FUNCTION_BLOCK FB_Clock
VAR_INPUT
	bStart : BOOL;
	bStop : BOOL;
	fCycleTime : LREAL;
END_VAR
VAR_OUTPUT
	fTime : LREAL;
END_VAR
VAR
END_VAR

IF bStart AND NOT(bStop) THEN
	fTime := fTime + fCycleTime;
ELSE
	fTime := 0.0;
END_IF

END_FUNCTION_BLOCK

(* stored: Version 1.1.0.1, ProductVersion 3.1.4024.9
   POU FB_Clock: Id {f13c44f0-374f-4488-b500-abcfceb96f9b}, SpecialFunc None *)
